DEF CloseNutGun(nutweldINFO :IN )
   ;FOLD Details
      ;FOLD Declaration
         DECL NutWeldDAT nutweldINFO
         BOOL bSkipGunChk, bSkipNutChk, bNutPresent, bMsgRelease
      ;ENDFOLD (Declaration)
      ;FOLD Implementation
         bSkipGunChk=FALSE
         bSkipNutChk=FALSE
         bNutPresent=FALSE
         bMsgRelease=FALSE
         dopw_NutIntensify(nutweldINFO.GunNr,FALSE)
         IF (bNutWeldWOJoining==FALSE) THEN
            dopw_GunWork(nutweldINFO.GunNr,TRUE)
            CONTINUE
            IF NOT (bSavedCurrentValue1 AND bSavedCurrentValue2 AND bSavedCurrentValue3) THEN
               SWITCH nutweldINFO.GunNr
                  CASE 1
                     IF NOT bSavedCurrentValue1 THEN
                        WAIT FOR bSavedCurrentValue1
                        rSetUpperLVDT_CLS_W_NUT[1] = aipw1_LVDT
                        rSetLowerLVDT_CLS_W_NUT[1] = aiNutSensorPW1
                        bSavedCurrentValue1        = TRUE
                     ENDIF
                  CASE 2
                     IF NOT bSavedCurrentValue2 THEN
                        WAIT FOR bSavedCurrentValue2
                        rSetUpperLVDT_CLS_W_NUT[2] = aipw2_LVDT
                        rSetLowerLVDT_CLS_W_NUT[2] = aiNutSensorPW2
                        bSavedCurrentValue2        = TRUE
                     ENDIF
                  CASE 3
                     IF NOT bSavedCurrentValue3 THEN
                        WAIT FOR bSavedCurrentValue3
                        rSetUpperLVDT_CLS_W_NUT[3] = aipw3_LVDT
                        rSetLowerLVDT_CLS_W_NUT[3] = aiNutSensorPW3
                        bSavedCurrentValue3        = TRUE
                     ENDIF
               ENDSWITCH
            ENDIF
            ;FOLD Gun Check
               $TIMER_STOP[nNutWeldSignalTmr]=TRUE
               $TIMER[nNutWeldSignalTmr]=nNutWeld_Signal_Timeout*(-1)
               $TIMER_STOP[nNutWeldSignalTmr]=FALSE
               WAIT FOR (((bpw_GunAtHome(nutweldINFO.GunNr)==FALSE) AND (bpw_GunAtWork(nutweldINFO.GunNr)==TRUE)) OR ($TIMER_FLAG[nNutWeldSignalTmr]==TRUE))
               $TIMER_STOP[nNutWeldSignalTmr]=TRUE
               IF (((bpw_GunAtHome(nutweldINFO.GunNr) == TRUE) OR (bpw_GunAtWork(nutweldINFO.GunNr) == FALSE)) AND (nDumpNutRetries <= nMaxDumpNutRetries)) THEN
                  bDump_Nut = TRUE
                  eCurrentState=#ERRORCloseGun
               ENDIF
               WHILE ((bNutWeldWOJoining==FALSE) AND ((bpw_GunAtHome(nutweldINFO.GunNr)==TRUE) OR (bpw_GunAtWork(nutweldINFO.GunNr)==FALSE)) AND (bSkipGunChk==FALSE) AND (nDumpNutRetries > nMaxDumpNutRetries))
                  ;FOLD Dialog "Nut Welder Open Switch Fault?"
                     REPEAT
                        nNutWeld_Handle = Set_KrlDlg (NutWeld_Msg[10], NutWeld_MsgPar[], NutWeld_SK_RetrySkip[], NutWeld_MsgOpt_Stop)
                        IF (nNutWeld_Handle > 0) THEN
                           WHILE (Exists_KrlDlg(nNutWeld_Handle, nNutWeld_Key))
                              WAIT SEC 0.024
                           ENDWHILE
                           SWITCH nNutWeld_Key
                              CASE 1 ; Diagnostic
                                 nNutWeld_Handle = Set_Krlmsg (#QUIT, NutWeld_Msg[2], NutWeld_MsgPar[], NutWeld_MsgOpt_Stop)
                                 WHILE (Exists_KrlMsg(nNutWeld_Handle))
                                    WAIT SEC 0.024
                                 ENDWHILE
                              CASE 2 ; Retry
                                 dopw_GunWork(nutweldINFO.GunNr,FALSE)
                                 WAIT SEC 1.0
                                 dopw_GunWork(nutweldINFO.GunNr,TRUE)
                                 $TIMER_STOP[nNutWeldSignalTmr]=TRUE
                                 $TIMER[nNutWeldSignalTmr]=nNutWeld_Signal_Timeout*(-1)
                                 $TIMER_STOP[nNutWeldSignalTmr]=FALSE
                                 WAIT FOR (((bpw_GunAtHome(nutweldINFO.GunNr)==FALSE) AND (bpw_GunAtWork(nutweldINFO.GunNr)==TRUE)) OR ($TIMER_FLAG[nNutWeldSignalTmr]==TRUE))
                                 $TIMER_STOP[nNutWeldSignalTmr]=TRUE
                                 bMsgRelease=TRUE
                              CASE 3 ; Skip
                                 WAIT SEC 0.100
                                 bMsgRelease=TRUE
                                 bSkipGunChk=TRUE
                           ENDSWITCH
                        ENDIF
                     UNTIL (bMsgRelease==TRUE)
                     bMsgRelease=FALSE
                  ;ENDFOLD (Dialog)
               ENDWHILE
            ;ENDFOLD (Gun Check)
            IF (PNWStyle==#STUDWELD) THEN
               dopw_StudStripped(nutweldINFO.GunNr,TRUE)
               dopw_StartFeed(nutweldINFO.GunNr,FALSE)
               ;FOLD Wait DI dipw_SpearHome==TRUE
                  $TIMER_STOP[nNutWeldSignalTmr]=TRUE
                  $TIMER[nNutWeldSignalTmr]=nNutWeld_Signal_Timeout*(-1)
                  $TIMER_STOP[nNutWeldSignalTmr]=FALSE
                  WAIT FOR ((dipw_SpearHome(nutweldINFO.GunNr)==TRUE) OR ($TIMER_FLAG[nNutWeldSignalTmr]==TRUE))
                  $TIMER_STOP[nNutWeldSignalTmr]=TRUE
               ;ENDFOLD (WaitDI dipw_SpearHome==TRUE)
            ENDIF
         ENDIF
      ;ENDFOLD (Implementation)
   ;ENDFOLD (Details)
END ; (CloseNutGun)

DEF CheckNutPresent(nutweldINFO :IN)
   ;FOLD Details
      ;FOLD Declaration
         DECL NutWeldDAT nutweldINFO
         DECL BOOL bNutChkComplete
         DECL BOOL bSkipNutChk
         DECL BOOL bInRetry
         DECL BOOL bMsgRelease
         DECL BOOL bToleranceWindowOK
         DECL REAL rSensorSample
         DECL REAL rLVDTSample
      ;ENDFOLD (Declaration)
      ;FOLD Implementation
         bMsgRelease=FALSE
         bNutChkComplete=FALSE
         bSkipNutChk=FALSE
         bInRetry=FALSE
         bToleranceWindowOK=FALSE
         WAIT FOR NOT bByPassSmartelec
         IF (bByPassSmartelec == TRUE) THEN
            RETURN ; Exit without checking
         ENDIF
         IF ((bNutWeldWOJoining==TRUE) OR (bPNWBlockFeed==TRUE)) THEN
            WAIT SEC 0.15
            RETURN ; Exit after check delay
         ENDIF
         nFeedRetries=0
         REPEAT
            bNutChkComplete=FALSE
            bInRetry=FALSE
            WAIT FOR ((rHighTolInUse-rLowTolInUse)>0) AND ((rHighTolInUse-rLowTolInUse)<1750)
            WAIT FOR ((rHighLVDTTolInUse-rLowLVDTTolInUse)>0) AND ((rHighLVDTTolInUse-rLowLVDTTolInUse)<1750)
            WAIT FOR ((rLowTolInUse)>0)
            WAIT FOR ((rHighTolInUse)>0)
            WAIT FOR ((rLowLVDTTolInUse)>0)
            WAIT FOR ((rHighLVDTTolInUse)>0)
            CloseNutGun(nutweldINFO)
            SensorSettle(nutweldINFO)
            rSensorSample=ABS(aiNutSensor(nutweldINFO.GunNr))   ; lower LVDT
            rLVDTSample=ABS(aiLVDTSensor(nutweldINFO.GunNr))    ; upper LVDT
            IF ((rSensorSample >= rLowTolInUse) AND (rSensorSample <= rHighTolInUse) AND (rLVDTSample >= rLowLVDTTolInUse) AND (rLVDTSample <= rHighLVDTTolInUse))  THEN
               bSkipNutChk=TRUE   ; do not check missing or inverted Nut if within range!
               ;save rSensorSample
               rNutSaveCount=rNutSaveCount+1
               IF (rNutSaveCount<1)OR (rNutSaveCount>50) THEN
                  rNutSaveCount=1
               ENDIF
               rNutSaveValue[rNutSaveCount]=rSensorSample
               rLVDTSaveValue[rNutSaveCount]=rLVDTSample
            ENDIF
            ;FOLD Nut Check Sequence
               ;FOLD Check for Inverted Nut
                  IF (((rSensorSample >= rHighTolInUse) OR (rLVDTSample < rLowLVDTTolInUse) OR (rLVDTSample > rHighLVDTTolInUse)) AND (nDumpNutRetries <= nMaxDumpNutRetries)) THEN
                     bDump_Nut=TRUE
                     eCurrentState=#ERRORInvertedNut
                     bNutChkComplete=FALSE
                  ENDIF
                  IF ((bSkipNutChk==FALSE) AND (bInRetry==FALSE) AND (nDumpNutRetries > nMaxDumpNutRetries)) THEN
                     IF ((rSensorSample >= rHighTolInUse) OR (rLVDTSample < rLowLVDTTolInUse) OR (rLVDTSample > rHighLVDTTolInUse)) THEN
                        ;FOLD Dialog "Nut Inverted Fault!  Press SKIP to Ignore Or Retry to Open and Close the Gun."
                           REPEAT
                              nNutWeld_Handle = Set_KrlDlg (NutWeld_Msg[48], NutWeld_MsgPar[], NutWeld_SK_RetrySkip[], NutWeld_MsgOpt_Stop)
                              IF (nNutWeld_Handle > 0) THEN
                                 WHILE (Exists_KrlDlg(nNutWeld_Handle, nNutWeld_Key))
                                    IF ($ERR.Int_Prio>0) THEN
                                       BRAKE
                                    ENDIF
                                    WAIT SEC 0.024
                                 ENDWHILE
                                 SWITCH nNutWeld_Key
                                    CASE 1 ; Diagnostic
                                       nNutWeld_Handle = Set_Krlmsg (#QUIT, NutWeld_Msg[2], NutWeld_MsgPar[], NutWeld_MsgOpt_Stop)
                                       WHILE (Exists_KrlMsg(nNutWeld_Handle))
                                          WAIT SEC 0.024
                                       ENDWHILE
                                    CASE 2 ; Retry
                                       bMsgRelease=TRUE
                                       bNutChkComplete=FALSE
                                       bInRetry=TRUE
                                       dopw_GunWork(nutweldINFO.GunNr,FALSE)
                                       WAIT SEC 1.5
                                       IF (($MODE_OP==#T1) OR ($MODE_OP==#T2)) THEN
                                          HALT
                                       ENDIF
                                    CASE 3 ; Skip
                                       WAIT SEC 0.100
                                       bMsgRelease=TRUE
                                       bSkipNutChk=TRUE
                                 ENDSWITCH
                              ENDIF
                           UNTIL (bMsgRelease==TRUE)
                           bMsgRelease=FALSE
                        ;ENDFOLD (Dialog)
                     ENDIF
                  ENDIF
               ;ENDFOLD (Check for Inverted Nut)
               ;FOLD Check for Nut Missing, If No Nut - Open Gun and feed new nut
                  IF ((bSkipNutChk==FALSE) AND (bInRetry==FALSE)) THEN
                     rSensorSample=ABS(aiNutSensor(nutweldINFO.GunNr))
                     IF ((rSensorSample <= rLowTolInUse) AND (nDumpNutRetries <= nMaxDumpNutRetries)) THEN
                        bDump_Nut=TRUE
                        eCurrentState=#ERRORNoNut
                        bNutChkComplete=FALSE
                     ENDIF
                     IF ((rSensorSample <= rLowTolInUse) AND (nDumpNutRetries > nMaxDumpNutRetries)) THEN
                        ;FOLD Dialog "Nut Not Detected Fault!  Press SKIP to Ignore Or Retry to Refeed a Nut."
                           REPEAT
                              nNutWeld_Handle = Set_KrlDlg (NutWeld_Msg[13], NutWeld_MsgPar[], NutWeld_SK_RetrySkip[], NutWeld_MsgOpt_Stop)
                              IF (nNutWeld_Handle > 0) THEN
                                 WHILE (Exists_KrlDlg(nNutWeld_Handle, nNutWeld_Key))
                                    IF ($ERR.Int_Prio>0) THEN
                                       BRAKE
                                    ENDIF
                                    WAIT SEC 0.024
                                 ENDWHILE
                                 SWITCH nNutWeld_Key
                                    CASE 1 ; Diagnostic
                                       nNutWeld_Handle = Set_Krlmsg (#QUIT, NutWeld_Msg[2], NutWeld_MsgPar[], NutWeld_MsgOpt_Stop)
                                       WHILE (Exists_KrlMsg(nNutWeld_Handle))
                                          WAIT SEC 0.024
                                       ENDWHILE
                                    CASE 2 ; Retry
                                       bMsgRelease=TRUE
                                       bNutChkComplete=FALSE
                                       bInRetry=TRUE
                                       nFeedRetries=0
                                       OpenNutGun(nutweldINFO)
                                       FeedNutReq(nutweldINFO)
                                    CASE 3 ; Skip
                                       WAIT SEC 0.100
                                       bSkipNutChk=TRUE
                                       bMsgRelease=TRUE
                                 ENDSWITCH
                              ENDIF
                           UNTIL (bMsgRelease==TRUE)
                           bMsgRelease=FALSE
                        ;ENDFOLD (Dialog)
                     ENDIF
                  ENDIF
               ;ENDFOLD (Check for Nut Missing, If No Nut - Open Gun and feed new nut)
            ;ENDFOLD (Nut Check Sequence)
         UNTIL ((bNutChkComplete==TRUE)  OR  (bSkipNutChk==TRUE) OR (bDump_Nut==TRUE))
      ;ENDFOLD (Implementation)
   ;ENDFOLD (Details)
END ; (CheckNutPresent)

;move to Reload position
GLOBAL DEF Nut_ToReloadPos(WeldPos:IN, WeldBase:IN, EnableReload:IN, Move1:IN, Move2:IN, Move3:IN, ReloadPos1:IN, ReloadPos2:IN, ReloadPos3:IN, ReloadBase1:IN, ReloadBase2:IN, ReloadBase3:IN)
   INT EnableReload
   E6POS WeldPos,ReloadPos1,ReloadPos2,ReloadPos3
   DECL FDAT WeldBase,ReloadBase1,ReloadBase2,ReloadBase3
   DECL Nut_Dump_Move Move1,Move2,Move3

   SWITCH (EnableReload)
      CASE 1
         Nut_ReLoad(Move1,ReloadPos1,ReloadBase1,FALSE)
      CASE 2
         Nut_ReLoad(Move1,ReloadPos1,ReloadBase1,FALSE)
         Nut_ReLoad(Move2,ReloadPos2,ReloadBase2,FALSE)
      CASE 3
         Nut_ReLoad(Move1,ReloadPos1,ReloadBase1,FALSE)
         Nut_ReLoad(Move2,ReloadPos2,ReloadBase2,TRUE)
         Nut_ReLoad(Move3,ReloadPos3,ReloadBase3,FALSE)
   ENDSWITCH
   WAIT FOR $IN[1025]

END

;move to Weld position
GLOBAL DEF Nut_ToWeldPos(WeldPos:IN, WeldBase:IN, EnableReload:IN, Move1:IN, Move2:IN, Move3:IN, ReloadPos1:IN, ReloadPos2:IN, ReloadPos3:IN, ReloadBase1:IN, ReloadBase2:IN, ReloadBase3:IN)
   INT EnableReload
   E6POS WeldPos,ReloadPos1,ReloadPos2,ReloadPos3
   DECL FDAT WeldBase,ReloadBase1,ReloadBase2,ReloadBase3
   DECL Nut_Dump_Move Move1,Move2,Move3

   SWITCH (EnableReload)
      CASE 1
         Nut_ReLoad(Move1,WeldPos,WeldBase,FALSE)
      CASE 2
         Nut_ReLoad(Move2,ReloadPos1,ReloadBase1,TRUE)
         Nut_ReLoad(Move1,WeldPos,WeldBase,FALSE)
      CASE 3
         Nut_ReLoad(Move3,ReloadPos2,ReloadBase2,TRUE)
         Nut_ReLoad(Move2,ReloadPos1,ReloadBase1,TRUE)
         Nut_ReLoad(Move1,WeldPos,WeldBase,FALSE)
   ENDSWITCH
   WAIT FOR $IN[1025]

END

;only for move to Reload Pos at block selection
GLOBAL DEF Nut_ReloadPos(Move1:IN, ReloadPos:IN)
   E6POS ReloadPos
   DECL Nut_Dump_Move Move1

   IF ($Mode_OP==#T1)THEN
      IF ($MOVE_BCO) THEN
         nNutWeld_Handle_SPS=Set_Krlmsg (#NOTIFY, NutWeld_Msg[61], NutWeld_MsgPar[], NutWeld_MsgOpt_NoStop)
         IF Move1==#Reload_PTP THEN
            PTP ReloadPos
         ELSE
            LIN ReloadPos
         ENDIF
         nNutWeld_Handle_SPS=Set_Krlmsg (#NOTIFY, NutWeld_Msg[62], NutWeld_MsgPar[], NutWeld_MsgOpt_NoStop)
      ENDIF
   ENDIF

END

GLOBAL DEF Nut_ReLoad(Drive:IN, ReloadPos:IN, ReloadBase:IN, Cont:IN)
   E6POS ReloadPos
   DECL FDAT ReloadBase
   DECL Nut_Dump_Move Drive
   BOOL Cont

   IF Drive==#Reload_PTP THEN
      PDAT_ACT=nut_PRELOAD
      FDAT_ACT=ReloadBase
      BAS(#PTP_PARAMS,nut_PRELOAD.VEL)
      IF Cont THEN
         PTP ReloadPos C_DIS
      ELSE
         PTP ReloadPos
      ENDIF
   ELSE ;#Reload_LIN
      LDAT_ACT=nut_LCRELOAD
      FDAT_ACT=ReloadBase
      BAS(#CP_PARAMS,nut_LCRELOAD.VEL)
      IF Cont THEN
         LIN ReloadPos C_DIS C_DIS
      ELSE
         LIN ReloadPos
      ENDIF
   ENDIF

END

DEF IntensfNutGun(nutweldINFO :IN )
   ;FOLD Details
      ;FOLD Declaration
         DECL NutWeldDAT nutweldINFO
         DECL BOOL bMsgRelease
         DECL BOOL bPreChkSkp
         DECL BOOL bIntensfChkSkp
      ;ENDFOLD (Declaration)
      ;FOLD Implementation
         bMsgRelease=FALSE
         bPreChkSkp=FALSE
         bIntensfChkSkp=FALSE
         IF (bNutWeldWOJoining==FALSE) THEN
            ;FOLD TimeOut Setup
               $TIMER_STOP[nNutWeldSignalTmr]=TRUE
               $TIMER[nNutWeldSignalTmr]=nNutWeld_Signal_Timeout*(-1)
               $TIMER_STOP[nNutWeldSignalTmr]=FALSE
            ;ENDFOLD (TimeOut Setup)
            WAIT FOR ((dipw_IntensfPresOk(nutweldINFO.GunNr)==FALSE) OR ($TIMER_FLAG[nNutWeldSignalTmr]==TRUE))
            $TIMER_STOP[nNutWeldSignalTmr]=TRUE
            WHILE ((dipw_IntensfPresOk(nutweldINFO.GunNr)==TRUE) AND (bPreChkSkp==FALSE))
               ;FOLD Dialog "Nut Welder Intensify Pressure Fault!  Pressure Switch Remained On From Last Cycle!"
                  REPEAT
                     nNutWeld_Handle = Set_KrlDlg (NutWeld_Msg[17], NutWeld_MsgPar[], NutWeld_SK_RetrySkip[], NutWeld_MsgOpt_Stop)
                     IF (nNutWeld_Handle > 0) THEN
                        WHILE (Exists_KrlDlg(nNutWeld_Handle, nNutWeld_Key))
                           IF ($ERR.Int_Prio>0) THEN
                              BRAKE
                           ENDIF
                           WAIT SEC 0.024
                        ENDWHILE
                        SWITCH nNutWeld_Key
                           CASE 1 ; Diagnostic
                              nNutWeld_Handle = Set_Krlmsg (#QUIT, NutWeld_Msg[2], NutWeld_MsgPar[], NutWeld_MsgOpt_Stop)
                              WHILE (Exists_KrlMsg(nNutWeld_Handle))
                                 WAIT SEC 0.024
                              ENDWHILE
                           CASE 2 ; Retry
                              bMsgRelease=TRUE
                           CASE 3 ; Skip
                              WAIT SEC 0.100
                              bMsgRelease=TRUE
                              bPreChkSkp=TRUE
                        ENDSWITCH
                     ENDIF
                  UNTIL (bMsgRelease==TRUE)
                  bMsgRelease=FALSE
               ;ENDFOLD (Dialog)
            ENDWHILE
            dopw_BlowOff(nutweldINFO.GunNr,TRUE)
            dopw_StudStripped(nutweldINFO.GunNr,FALSE)
            dopw_NutIntensify(nutweldINFO.GunNr, TRUE)
            ;FOLD TimeOut Setup
               $TIMER_STOP[nNutWeldSignalTmr]=TRUE
               $TIMER[nNutWeldSignalTmr]=nNutWeld_Signal_Timeout*(-1)
               $TIMER_STOP[nNutWeldSignalTmr]=FALSE
               WAIT FOR ((dipw_IntensfPresOk(nutweldINFO.GunNr)==TRUE) OR ($TIMER_FLAG[nNutWeldSignalTmr]==TRUE))
               $TIMER_STOP[nNutWeldSignalTmr]=TRUE
               WHILE ((dipw_IntensfPresOk(nutweldINFO.GunNr)==FALSE) AND (bIntensfChkSkp==FALSE))
                  ;FOLD Dialog "Nut Welder Intensify Pressure Fault!  Pressure Switch Is Not On!"
                     eCurrentState=#ERRORIntensifyWelder
                     REPEAT
                        nNutWeld_Handle = Set_KrlDlg (NutWeld_Msg[18], NutWeld_MsgPar[], NutWeld_SK_RetrySkip[], NutWeld_MsgOpt_Stop)
                        IF (nNutWeld_Handle > 0) THEN
                           WHILE (Exists_KrlDlg(nNutWeld_Handle, nNutWeld_Key))
                              IF ($ERR.Int_Prio>0) THEN
                                 BRAKE
                              ENDIF
                              WAIT SEC 0.024
                           ENDWHILE
                           SWITCH nNutWeld_Key
                              CASE 1 ; Diagnostic
                                 nNutWeld_Handle = Set_Krlmsg (#QUIT, NutWeld_Msg[2], NutWeld_MsgPar[], NutWeld_MsgOpt_Stop)
                                 WHILE (Exists_KrlMsg(nNutWeld_Handle))
                                    WAIT SEC 0.024
                                 ENDWHILE
                              CASE 2 ; Retry
                                 bMsgRelease=TRUE
                              CASE 3 ; Skip
                                 WAIT SEC 0.100
                                 bMsgRelease=TRUE
                                 bIntensfChkSkp=TRUE
                           ENDSWITCH
                        ENDIF
                     UNTIL (bMsgRelease==TRUE)
                     bMsgRelease=FALSE
                  ;ENDFOLD (Dialog)
               ENDWHILE

            ;ENDFOLD (TimeOut Setup)
         ENDIF
      ;ENDFOLD (Implementation)
   ;ENDFOLD (Details)
END ; (IntensfNutGun)

DEF WeldInitiate(nutweldINFO :IN )
   ;FOLD Details
      ;FOLD Declaration
         DECL NutWeldDAT nutweldINFO
         DECL BOOL bSkipWeld
         DECL BOOL bWeldComplete
         DECL BOOL bMsgRelease
      ;ENDFOLD (Declaration)
      ;FOLD Implementation
         bMsgRelease=FALSE
         bSkipWeld=FALSE
         ;FOLD Check the Water Flow
            WHILE NOT (di474WaterOk OR di522WaterOk OR di570WaterOk)
               IF NOT di474WaterOk THEN
                  $LOOP_MSG[] = " No WaterFlow in Gun1                                                                                                  "
               ENDIF
               IF NOT di522WaterOk THEN
                  $LOOP_MSG[] = " No WaterFlow in Gun2                                                                                                  "
               ENDIF
               IF NOT di570WaterOk THEN
                  $LOOP_MSG[] = " No WaterFlow in Gun3                                                                                                  "
               ENDIF
            ENDWHILE
            $LOOP_MSG[] = "                                                                                                                    "
         ;ENDFOLD (Check the Water Flow )
         ;FOLD Check the Temperature Water
            WHILE NOT (di472WaterTempOK OR di520WaterTempOK OR di568WaterTempOK)
               IF NOT di472WaterTempOK THEN
                  $LOOP_MSG[] = " No WaterTemp in Gun1                                                                                                  "
               ENDIF
               IF NOT di520WaterTempOK THEN
                  $LOOP_MSG[] = " No WaterTemp in Gun2                                                                                                  "
               ENDIF
               IF NOT di568WaterTempOK THEN
                  $LOOP_MSG[] = " No WaterTemp in Gun3                                                                                                  "
               ENDIF
            ENDWHILE
            $LOOP_MSG[] = "                                                                                                                    "
         ;ENDFOLD (Check the Temperature Water)
         IF (bNutWeld_InhibitWeld==TRUE) THEN
            RETURN
         ENDIF
         IF (bNutWeldWOJoining==FALSE) THEN
            REPEAT
               bWeldComplete=TRUE
               $TIMER_STOP[nNutWeldSignalTmr]=TRUE
               $TIMER[nNutWeldSignalTmr]=nNutWeld_Weld_Timeout*(-1000)
               $TIMER_STOP[nNutWeldSignalTmr]=FALSE
               dopw_WeldInit(nutweldINFO.GunNr,TRUE)
               WAIT FOR ((dipw_WeldComplete(nutweldINFO.GunNr)==TRUE) OR ($TIMER_FLAG[nNutWeldSignalTmr]==TRUE))
               $TIMER_STOP[nNutWeldSignalTmr]=TRUE

               IF (dipw_WeldComplete(nutweldINFO.GunNr)) THEN   ;count 1 weld up
                  AC_Process_Count(#Count1up)
               ENDIF

               IF ((dipw_WeldComplete(nutweldINFO.GunNr)==FALSE)) THEN
                  dopw_WeldInit(nutweldINFO.GunNr,FALSE)
                  bWeldComplete=FALSE
                  nWeldRetries = nWeldRetries + 1
                  IF (nWeldRetries > nMaxWeldRetries) then
                     do004ProcessFault=TRUE
                     ;FOLD Dialog "WELD NOT COMPLETE! Mark part as scrap, scrap part at end of cycle"
                        REPEAT
                           nNutWeld_Handle = Set_KrlDlg (NutWeld_Msg[19], NutWeld_MsgPar[], NutWeld_SK_OK[], NutWeld_MsgOpt_Stop)
                           IF (nNutWeld_Handle > 0) THEN
                              WHILE (Exists_KrlDlg(nNutWeld_Handle, nNutWeld_Key))
                                 WAIT SEC 0.024
                              ENDWHILE
                              SWITCH nNutWeld_Key
                                 CASE 1 ; Skip
                                    bWeldComplete=FALSE
                                    bMsgRelease=TRUE
                                    bSkipWeld=TRUE
                              ENDSWITCH
                              do004ProcessFault=FALSE
                           ENDIF
                        UNTIL (bMsgRelease==TRUE)
                        bMsgRelease=FALSE
                     ;ENDFOLD (Dialog)
                  ENDIF
               ENDIF
            UNTIL ((bWeldComplete==TRUE) OR (bSkipWeld==TRUE))
            bSkipWeld=FALSE
         ENDIF
         dopw_WeldInit(nutweldINFO.GunNr,FALSE)
      ;ENDFOLD (Implementation)
   ;ENDFOLD (Details)
END ; (WeldInitiate)

DEF FeedNutReq(nutweldINFO :IN)
   ;FOLD Details
      ;FOLD Declaration
         DECL NutWeldDAT nutweldINFO
         DECL BOOL bSkipPinRet
         DECL BOOL bMsgRelease
         DECL BOOL bSkipFeed
      ;ENDFOLD (Declaration)
      ;FOLD Implementation
         bSkipPinRet=FALSE
         bMsgRelease=FALSE
         bSkipFeed=FALSE
         IF ((bNutWeldWOJoining==TRUE) OR (bPNWBlockFeed==TRUE)) THEN
            WAIT SEC 0.15
            RETURN ; Exit after check delay
         ENDIF
         ;FOLD Check that the Locate Pin is Advanced
            dopw_PinAdv(nutweldINFO.GunNr, TRUE)
            $TIMER_STOP[nNutWeldSignalTmr]=TRUE
            $TIMER[nNutWeldSignalTmr]=nNutWeld_Signal_Timeout*(-1)
            $TIMER_STOP[nNutWeldSignalTmr]=FALSE
            WAIT FOR ((dipw_PinReturn(nutweldINFO.GunNr)==FALSE) OR ($TIMER_FLAG[nNutWeldSignalTmr]==TRUE)) ; Convert to no nut analog
            $TIMER_STOP[nNutWeldSignalTmr]=TRUE
            ; Modified for nutweld specific, original refernce was studweld
            WHILE ((dipw_PinReturn(nutweldINFO.GunNr)==TRUE) AND (bSkipPinRet==FALSE))
               ;FOLD Dialog "Welder Pin is Not Advanced!  Check the Pin or Smart Electrode!"
                  REPEAT
                     nNutWeld_Handle = Set_KrlDlg (NutWeld_Msg[15], NutWeld_MsgPar[], NutWeld_SK_RetrySkip[], NutWeld_MsgOpt_Stop)
                     IF (nNutWeld_Handle > 0) THEN
                        WHILE (Exists_KrlDlg(nNutWeld_Handle, nNutWeld_Key))
                           WAIT SEC 0.024
                        ENDWHILE
                        SWITCH nNutWeld_Key
                           CASE 1 ; Diagnostic
                              nNutWeld_Handle = Set_Krlmsg (#QUIT, NutWeld_Msg[2], NutWeld_MsgPar[], NutWeld_MsgOpt_Stop)
                              WHILE (Exists_KrlMsg(nNutWeld_Handle))
                                 WAIT SEC 0.024
                              ENDWHILE
                           CASE 2 ; Retry
                              bMsgRelease=TRUE
                           CASE 3 ; Skip
                              bMsgRelease=TRUE
                              bSkipPinRet=TRUE
                        ENDSWITCH
                     ENDIF
                  UNTIL (bMsgRelease==TRUE)
                  bMsgRelease=FALSE
               ;ENDFOLD (Dialog)
            ENDWHILE
         ;ENDFOLD (Check that the Locate Pin is Advanced)
         dopw_StartFeed(nutweldINFO.GunNr,TRUE)
         ;FOLD WaitDI dipw_SpearHome==FALSE
            $TIMER_STOP[nNutWeldSignalTmr]=TRUE
            $TIMER[nNutWeldSignalTmr]=nNutWeld_Signal_Timeout*(-1)
            $TIMER_STOP[nNutWeldSignalTmr]=FALSE
            WAIT FOR ((dipw_SpearHome(nutweldINFO.GunNr)==FALSE) OR ($TIMER_FLAG[nNutWeldSignalTmr]==TRUE))
            $TIMER_STOP[nNutWeldSignalTmr]=TRUE
         ;ENDFOLD (WaitDI dipw_SpearHome==FALSE)
         IF (PNWStyle==#NUTWELD) THEN
            ;FOLD WaitDI dipw_SpearHome==TRUE
               $TIMER_STOP[nNutWeldSignalTmr]=TRUE
               $TIMER[nNutWeldSignalTmr]=nNutWeld_Signal_Timeout*(-1)
               $TIMER_STOP[nNutWeldSignalTmr]=FALSE
               WAIT FOR ((dipw_SpearHome(nutweldINFO.GunNr)==TRUE) OR ($TIMER_FLAG[nNutWeldSignalTmr]==TRUE))
               $TIMER_STOP[nNutWeldSignalTmr]=TRUE
            ;ENDFOLD (WaitDI dipw_SpearHome==TRUE)
         ENDIF
         ;FOLD WaitDI dipw_FeedComplt==TRUE
            $TIMER_STOP[nNutWeldFeedTmr]=TRUE
            $TIMER[nNutWeldFeedTmr]=nNutWeld_Feed_Timeout*(-3000)
            $TIMER_STOP[nNutWeldFeedTmr]=FALSE
            WAIT FOR ((dipw_FeedComplt(nutweldINFO.GunNr)==TRUE) OR ($TIMER_FLAG[nNutWeldFeedTmr]==TRUE))
            $TIMER_STOP[nNutWeldFeedTmr]=TRUE
            WHILE ((dipw_FeedComplt(nutweldINFO.GunNr)==FALSE) AND (bSkipFeed==FALSE))
               ;FOLD Dialog "Feed Request Timeout Fault!  Check the Bowl Feeder!"
                  REPEAT
                     nNutWeld_Handle = Set_KrlDlg (NutWeld_Msg[49], NutWeld_MsgPar[], NutWeld_SK_RetrySkip[], NutWeld_MsgOpt_Stop)
                     IF (nNutWeld_Handle > 0) THEN
                        WHILE (Exists_KrlDlg(nNutWeld_Handle, nNutWeld_Key))
                           WAIT SEC 0.024
                        ENDWHILE
                        SWITCH nNutWeld_Key
                           CASE 1 ; Diagnostic
                              nNutWeld_Handle = Set_Krlmsg (#QUIT, NutWeld_Msg[2], NutWeld_MsgPar[], NutWeld_MsgOpt_Stop)
                              WHILE (Exists_KrlMsg(nNutWeld_Handle))
                                 WAIT SEC 0.024
                              ENDWHILE
                           CASE 2 ; Retry
                              bMsgRelease=TRUE
                              dopw_StartFeed(nutweldINFO.GunNr,FALSE)
                              WAIT SEC 1
                              dopw_StartFeed(nutweldINFO.GunNr,TRUE)
                              WAIT SEC 2
                           CASE 3 ; Skip
                              bMsgRelease=TRUE
                              bSkipFeed=TRUE
                        ENDSWITCH
                     ENDIF
                  UNTIL (bMsgRelease==TRUE)
                  bMsgRelease=FALSE
               ;ENDFOLD (Dialog)
            ENDWHILE
         ;ENDFOLD (WaitDI dipw_FeedComplt==TRUE)
         IF (PNWStyle==#NUTWELD) THEN
            dopw_StartFeed(nutweldINFO.GunNr,FALSE)
         ENDIF
      ;ENDFOLD (Implementation)
   ;ENDFOLD (Details)
END ; (FeedNutReq)

DEF SensorSettle(nutweldINFO :IN )
   ;FOLD Details
      ;FOLD Declaration
         DECL NutWeldDAT nutweldINFO
         REAL rPrimaryValue, rSecondaryValue, rSensorSample
      ;ENDFOLD (Declaration)
      ;FOLD Implementation
         REPEAT
            rPrimaryValue = ABS(aiNutSensor(nutweldINFO.GunNr))
            WAIT SEC rSensorSettleTime
            rSecondaryValue = ABS(aiNutSensor(nutweldINFO.GunNr))
            IF (ABS(rPrimaryValue - rSecondaryValue) > 40) THEN
               WAIT SEC rSensorSettleTime
            ENDIF
         UNTIL (ABS(rPrimaryValue - rSecondaryValue)<20)
      ;ENDFOLD (Implementation)
   ;ENDFOLD (Details)
END ; (SensorSettle)

DEF dopw_NutIntensify(nGunNr :IN, bState :IN )
   ;FOLD Details
      ;FOLD Declaration
         DECL INT nGunNr
         DECL BOOL bState
      ;ENDFOLD (Declaration)
      ;FOLD Implementation
         SWITCH nGunNr
            CASE 1
               dopw1_Nut1Intensify_Home=NOT(bState)
               dopw1_Nut1Intensify=bState
            CASE 2
               dopw2_Nut1Intensify_Home=NOT(bState)
               dopw2_Nut1Intensify=bState
            CASE 3
               dopw3_Nut1Intensify_Home=NOT(bState)
               dopw3_Nut1Intensify=bState
         ENDSWITCH
      ;ENDFOLD (Implementation)
   ;ENDFOLD (Details)
END ; (dopw_NutIntensify)

DEF dopw_GunWork(nGunNr :IN, bState :IN )
   ;FOLD Details
      ;FOLD Declaration
         DECL INT nGunNr
         DECL BOOL bState
      ;ENDFOLD (Declaration)
      ;FOLD Implementation
         SWITCH nGunNr
            CASE 1
               dopw1_GunWork=bState
               dopw1_GunHome=NOT (bState)
               IF (bState==FALSE) THEN
                  dopw_NutIntensify(nGunNr,FALSE)
               ENDIF
            CASE 2
               dopw2_GunWork=bState
               dopw2_GunHome=NOT (bState)
               IF (bState==FALSE) THEN
                  dopw_NutIntensify(nGunNr,FALSE)
               ENDIF
            CASE 3
               dopw3_GunWork=bState
               dopw3_GunHome=NOT (bState)
               IF (bState==FALSE) THEN
                  dopw_NutIntensify(nGunNr,FALSE)
               ENDIF
         ENDSWITCH
      ;ENDFOLD (Implementation)
   ;ENDFOLD (Details)
END ; (dopw_GunWork)

DEF dopw_PinAdv(nGunNr :IN, bState :IN )
   ;FOLD Details
      ;FOLD Declaration
         DECL INT nGunNr
         DECL BOOL bState
      ;ENDFOLD (Declaration)
      ;FOLD Implementation
         SWITCH nGunNr
            CASE 1
               dopw1_AdvancePin=bState
               dopw1_ReturnPin=NOT (bState)
            CASE 2
               dopw2_AdvancePin=bState
               dopw2_ReturnPin=NOT (bState)
            CASE 3
               dopw3_AdvancePin=bState
               dopw3_ReturnPin=NOT (bState)
         ENDSWITCH
      ;ENDFOLD (Implementation)
   ;ENDFOLD (Details)
END ; (dopw_PinAdv)

DEF dopw_StepperWarningPL(nGunNr :IN, bState :IN )
   ;FOLD Details
      ;FOLD Declaration
         DECL INT nGunNr
         DECL BOOL bState
      ;ENDFOLD (Declaration)
      ;FOLD Implementation
         SWITCH nGunNr
            CASE 1
               dopw1_StepperWarningPL=bState
            CASE 2
               dopw2_StepperWarningPL=bState
            CASE 3
               dopw3_StepperWarningPL=bState
         ENDSWITCH
      ;ENDFOLD (Implementation)
   ;ENDFOLD (Details)
END ; (dopw_StepperWarningPL)

DEF dopw_EndofStepperPL(nGunNr :IN, bState :IN )
   ;FOLD Details
      ;FOLD Declaration
         DECL INT nGunNr
         DECL BOOL bState
      ;ENDFOLD (Declaration)
      ;FOLD Implementation
         SWITCH nGunNr
            CASE 1
               dopw1_EndofStepperPL=bState
            CASE 2
               dopw2_EndofStepperPL=bState
            CASE 3
               dopw3_EndofStepperPL=bState
         ENDSWITCH
      ;ENDFOLD (Implementation)
   ;ENDFOLD (Details)
END ; (dopw_EndofStepperPL)

DEF dopw_StartFeed(nGunNr :IN, bState :IN )
   ;FOLD Details
      ;FOLD Declaration
         DECL INT nGunNr
         DECL BOOL bState
      ;ENDFOLD (Declaration)
      ;FOLD Implementation
         SWITCH nGunNr
            CASE 1
               dopw1_StartFeed=bState
            CASE 2
               dopw2_StartFeed=bState
            CASE 3
               dopw3_StartFeed=bState
         ENDSWITCH
      ;ENDFOLD (Implementation)
   ;ENDFOLD (Details)
END ; (dopw_StartFeed)

DEF dopw_StartWater(nGunNr :IN, bState :IN )
   ;FOLD Details
      ;FOLD Declaration
         DECL INT nGunNr
         DECL BOOL bState
      ;ENDFOLD (Declaration)
      ;FOLD Implementation
         SWITCH nGunNr
            CASE 1
               dopw1_StartWater=bState
            CASE 2
               dopw2_StartWater=bState
            CASE 3
               dopw3_StartWater=bState
         ENDSWITCH
      ;ENDFOLD (Implementation)
   ;ENDFOLD (Details)
END ; (dopw_StartWater)

DEF dopw_SetPrgNr(nGunNr :IN, nPrgNr :IN )
   ;FOLD Details
      ;FOLD Declaration
         DECL INT nGunNr
         DECL INT nPrgNr
      ;ENDFOLD (Declaration)
      ;FOLD Implementation
         SWITCH nGunNr
            CASE 1
               gdopw1_SpotNumber=nPrgNr
            CASE 2
               gdopw2_SpotNumber=nPrgNr
            CASE 3
               gdopw3_SpotNumber=nPrgNr
         ENDSWITCH
      ;ENDFOLD (Implementation)
   ;ENDFOLD (Details)
END ; (dopw_SetPrgNr)

DEF dopw_WeldInit(nGunNr :IN, bState :IN )
   ;FOLD Details
      ;FOLD Declaration
         DECL INT nGunNr
         DECL BOOL bState
      ;ENDFOLD (Declaration)
      ;FOLD Implementation
         SWITCH nGunNr
            CASE 1
               dopw1_WeldInit=bState
            CASE 2
               dopw2_WeldInit=bState
            CASE 3
               dopw3_WeldInit=bState
         ENDSWITCH
      ;ENDFOLD (Implementation)
   ;ENDFOLD (Details)
END ; (dopw_WeldInit)

DEF dopw_FaultReset(nGunNr :IN, bState :IN )
   ;FOLD Details
      ;FOLD Declaration
         DECL INT nGunNr
         DECL BOOL bState
      ;ENDFOLD (Declaration)
      ;FOLD Implementation
         SWITCH nGunNr
            CASE 1
               dopw1_FaultReset=bState
            CASE 2
               dopw2_FaultReset=bState
            CASE 3
               dopw3_FaultReset=bState
         ENDSWITCH
      ;ENDFOLD (Implementation)
   ;ENDFOLD (Details)
END ; (dopw_FaultReset)

DEF dopw_BlowOff(nGunNr :IN, bState :IN )
   ;FOLD Details
      ;FOLD Declaration
         DECL INT nGunNr
         DECL BOOL bState
      ;ENDFOLD (Declaration)
      ;FOLD Implementation
         SWITCH nGunNr
            CASE 1
               dopw1_BlowOff=bState
            CASE 2
               dopw2_BlowOff=bState
            CASE 3
               dopw3_BlowOff=bState
         ENDSWITCH
      ;ENDFOLD (Implementation)
   ;ENDFOLD (Details)
END ; (dopw_BlowOff)

DEF dopw_StudStripped(nGunNr :IN, bState :IN )
   ;FOLD Details
      ;FOLD Declaration
         DECL INT nGunNr
         DECL BOOL bState
      ;ENDFOLD (Declaration)
      ;FOLD Implementation
         SWITCH nGunNr
            CASE 1
               dopw1_StudStripped=bState
            CASE 2
               dopw2_StudStripped=bState
            CASE 3
               dopw3_StudStripped=bState
         ENDSWITCH
      ;ENDFOLD (Implementation)
   ;ENDFOLD (Details)
END ; (dopw_StudStripped)

DEFFCT INT Get_FaultResetNr(nGunNr :IN )
   ;FOLD Details
      ;FOLD Declaration
         DECL INT nGunNr
         DECL SIGINF SignalIOInfo
      ;ENDFOLD (Declaration)
      ;FOLD Implementation
         SWITCH nGunNr
            CASE 1
               SignalIOInfo=GET_SIG_INF("dopw1_FaultReset")
               RETURN(SignalIOInfo.IDX)
            CASE 2
               SignalIOInfo=GET_SIG_INF("dopw2_FaultReset")
               RETURN(SignalIOInfo.IDX)
            CASE 3
               SignalIOInfo=GET_SIG_INF("dopw3_FaultReset")
               RETURN(SignalIOInfo.IDX)
         ENDSWITCH
      ;ENDFOLD (Implementation)
   ;ENDFOLD (Details)
ENDFCT ; (Get_FaultResetNr)

DEFFCT BOOL bpw_GunAtHome(nGunNr :IN )
   ;FOLD Details
      ;FOLD Declaration
         DECL INT nGunNr
      ;ENDFOLD (Declaration)
      ;FOLD Implementation
         SWITCH nGunNr
            CASE 1
               RETURN(bpw1_GunAtHome)
            CASE 2
               RETURN(bpw2_GunAtHome)
            CASE 3
               RETURN(bpw3_GunAtHome)
         ENDSWITCH
      ;ENDFOLD (Implementation)
   ;ENDFOLD (Details)
ENDFCT ; (bpw_GunAtHome)

DEFFCT BOOL bpw_GunAtWork(nGunNr :IN )
   ;FOLD Details
      ;FOLD Declaration
         DECL INT nGunNr
      ;ENDFOLD (Declaration)
      ;FOLD Implementation
         $OUT[148]=FALSE
         SWITCH nGunNr
            CASE 1
               RETURN(bpw1_GunAtWork)
            CASE 2
               RETURN(bpw2_GunAtWork)
            CASE 3
               RETURN(bpw3_GunAtWork)
         ENDSWITCH
      ;ENDFOLD (Implementation)
   ;ENDFOLD (Details)
ENDFCT ; (bpw_GunAtWork)

DEFFCT BOOL dipw_IntensfPresOk(nGunNr :IN )
   ;FOLD Details
      ;FOLD Declaration
         DECL INT nGunNr
      ;ENDFOLD (Declaration)
      ;FOLD Implementation
         SWITCH nGunNr
            CASE 1
               RETURN(dipw1_IntensfPresOk)
            CASE 2
               RETURN(dipw2_IntensfPresOk)
            CASE 3
               RETURN(dipw3_IntensfPresOk)
         ENDSWITCH
      ;ENDFOLD (Implementation)
   ;ENDFOLD (Details)
ENDFCT ; (dipw_IntensfPresOk)

DEFFCT BOOL dipw_StepperWarning(nGunNr :IN )
   ;FOLD Details
      ;FOLD Declaration
         DECL INT nGunNr
      ;ENDFOLD (Declaration)
      ;FOLD Implementation
         SWITCH nGunNr
            CASE 1
               RETURN(dipw1_StepperWarning)
            CASE 2
               RETURN(dipw2_StepperWarning)
            CASE 3
               RETURN(dipw3_StepperWarning)
         ENDSWITCH
      ;ENDFOLD (Implementation)
   ;ENDFOLD (Details)
ENDFCT ; (dipw_StepperWarning)

DEFFCT BOOL dipw_EndOfStepper(nGunNr :IN )
   ;FOLD Details
      ;FOLD Declaration
         DECL INT nGunNr
      ;ENDFOLD (Declaration)
      ;FOLD Implementation
         SWITCH nGunNr
            CASE 1
               RETURN(dipw1_EndOfStepper)
            CASE 2
               RETURN(dipw2_EndOfStepper)
            CASE 3
               RETURN(dipw3_EndOfStepper)
         ENDSWITCH
      ;ENDFOLD (Implementation)
   ;ENDFOLD (Details)
ENDFCT ; (dipw_EndOfStepper)

DEFFCT BOOL dipw_XtfmrTempOk(nGunNr :IN )
   ;FOLD Details
      ;FOLD Declaration
         DECL INT nGunNr
      ;ENDFOLD (Declaration)
      ;FOLD Implementation
         SWITCH nGunNr
            CASE 1
               RETURN(dipw1_XtfmrTempOk)
            CASE 2
               RETURN(dipw2_XtfmrTempOk)
            CASE 3
               RETURN(dipw3_XtfmrTempOk)
         ENDSWITCH
      ;ENDFOLD (Implementation)
   ;ENDFOLD (Details)
ENDFCT ; (dipw_XtfmrTempOk)

DEFFCT BOOL dipw_WaterOk(nGunNr :IN )
   ;FOLD Details
      ;FOLD Declaration
         DECL INT nGunNr
      ;ENDFOLD (Declaration)
      ;FOLD Implementation
         SWITCH nGunNr
            CASE 1
               RETURN(dipw1_WaterOk)
            CASE 2
               RETURN(dipw2_WaterOk)
            CASE 3
               RETURN(dipw3_WaterOk)
         ENDSWITCH
      ;ENDFOLD (Implementation)
   ;ENDFOLD (Details)
ENDFCT ; (dipw_WaterOk)

DEFFCT BOOL dipw_WaterTempOk(nGunNr :IN )
   ;FOLD Details
      ;FOLD Declaration
         DECL INT nGunNr
      ;ENDFOLD (Declaration)
      ;FOLD Implementation
         SWITCH nGunNr
            CASE 1
               RETURN(di472WaterTempOk)
            CASE 2
               RETURN(di520WaterTempOk)
            CASE 3
               RETURN(di568WaterTempOk)
         ENDSWITCH
      ;ENDFOLD (Implementation)
   ;ENDFOLD (Details)
ENDFCT ; (dipw_WaterTempOk)

DEFFCT BOOL dipw_WeldComplete(nGunNr :IN )
   ;FOLD Details
      ;FOLD Declaration
         DECL INT nGunNr
      ;ENDFOLD (Declaration)
      ;FOLD Implementation
         SWITCH nGunNr
            CASE 1
               RETURN(dipw1_WeldComplete)
            CASE 2
               RETURN(dipw2_WeldComplete)
            CASE 3
               RETURN(dipw3_WeldComplete)
         ENDSWITCH
      ;ENDFOLD (Implementation)
   ;ENDFOLD (Details)
ENDFCT ; (dipw_WeldComplete)

DEFFCT BOOL dipw_Ready(nGunNr :IN )
   ;FOLD Details
      ;FOLD Declaration
         DECL INT nGunNr
      ;ENDFOLD (Declaration)
      ;FOLD Implementation
         SWITCH nGunNr
            CASE 1
               RETURN(dipw1_Ready)
            CASE 2
               RETURN(dipw2_Ready)
            CASE 3
               RETURN(dipw3_Ready)
         ENDSWITCH
      ;ENDFOLD (Implementation)
   ;ENDFOLD (Details)
ENDFCT ; (dipw_Ready)

DEFFCT BOOL dipw_Fault(nGunNr :IN )
   ;FOLD Details
      ;FOLD Declaration
         DECL INT nGunNr
      ;ENDFOLD (Declaration)
      ;FOLD Implementation
         SWITCH nGunNr
            CASE 1
               RETURN(dipw1_Fault)
            CASE 2
               RETURN(dipw2_Fault)
            CASE 3
               RETURN(dipw3_Fault)
         ENDSWITCH
      ;ENDFOLD (Implementation)
   ;ENDFOLD (Details)
ENDFCT ; (dipw_Fault)

DEFFCT BOOL dipw_SpearHome(nGunNr :IN )
   ;FOLD Details
      ;FOLD Declaration
         DECL INT nGunNr
      ;ENDFOLD (Declaration)
      ;FOLD Implementation
         SWITCH nGunNr
            CASE 1
               RETURN(dipw1_SpearHome)
            CASE 2
               RETURN(dipw2_SpearHome)
            CASE 3
               RETURN(dipw3_SpearHome)
         ENDSWITCH
      ;ENDFOLD (Implementation)
   ;ENDFOLD (Details)
ENDFCT ; (dipw_SpearHome)

DEFFCT BOOL dipw_PinReturn(nGunNr :IN )
   ;FOLD Details
      ;FOLD Declaration
         DECL INT nGunNr
      ;ENDFOLD (Declaration)
      ;FOLD Implementation
         SWITCH nGunNr
            CASE 1
               RETURN(dipw1_PinReturn)
            CASE 2
               RETURN(dipw2_PinReturn)
            CASE 3
               RETURN(dipw3_PinReturn)
         ENDSWITCH
      ;ENDFOLD (Implementation)
   ;ENDFOLD (Details)
ENDFCT ; (dipw_PinReturn)

DEFFCT BOOL dipw_FeedComplt(nGunNr :IN )
   ;FOLD Details
      ;FOLD Declaration
         DECL INT nGunNr
      ;ENDFOLD (Declaration)
      ;FOLD Implementation
         SWITCH nGunNr
            CASE 1
               RETURN(dipw1_FeedComplt)
            CASE 2
               RETURN(dipw2_FeedComplt)
            CASE 3
               RETURN(dipw3_FeedComplt)
         ENDSWITCH
      ;ENDFOLD (Implementation)
   ;ENDFOLD (Details)
ENDFCT ; (dipw_FeedComplt)

DEFFCT REAL aiNutSensor(nGunNr :IN )
   ;FOLD Details
      ;FOLD Declaration
         DECL INT nGunNr
      ;ENDFOLD (Declaration)
      ;FOLD Implementation
         SWITCH nGunNr
            CASE 1
               RETURN(aiNutSensorPW1)
            CASE 2
               RETURN(aiNutSensorPW2)
            CASE 3
               RETURN(aiNutSensorPW3)
         ENDSWITCH
      ;ENDFOLD (Implementation)
   ;ENDFOLD (Details)
ENDFCT ; (aiNutSensor)

DEFFCT REAL aiLVDTSensor(nGunNr :IN )
   ;FOLD Details
      ;FOLD Declaration
         DECL INT nGunNr
      ;ENDFOLD (Declaration)
      ;FOLD Implementation
         SWITCH nGunNr
            CASE 1
               RETURN(aipw1_LVDT)
            CASE 2
               RETURN(aipw2_LVDT)
            CASE 3
               RETURN(aipw3_LVDT)
         ENDSWITCH
      ;ENDFOLD (Implemenation)
   ;ENDFOLD (Details)
ENDFCT ; (aiLVDTSensor)

--- nutweldroutines.dat ---
&ACCESS RVO3
&REL 3482
&PARAM DISKPATH = KRC:\R1\TP\NutWeld
DEFDAT  nutweldroutines PUBLIC
;*********************************
;* Package:     NutWeldRoutines  *
;* Release      V1.0.4           *
;* Date:        01.2016          *
;* GUI Version: > = V8.3         *
;*********************************

GLOBAL ENUM Nut_Dump_Move Reload_PTP,Reload_LIN
DECL GLOBAL BOOL bDump_Nut
DECL GLOBAL INT nMaxGunNr=3
DECL GLOBAL INT nMaxWeldRetries=0
DECL GLOBAL INT nMaxFeedRetries=0
DECL GLOBAL INT nMaxDumpNutRetries=10
DECL GLOBAL INT nSpotNrTstCrnt=255
DECL GLOBAL BOOL bPNWBlockFeed=FALSE
DECL GLOBAL INT nNutWeldSignalTmr=41
DECL GLOBAL INT nNutWeld_Signal_Timeout=6000 ; (ms)
DECL GLOBAL INT nNutWeldFeedTmr=41
DECL GLOBAL INT nNutWeld_Feed_Timeout=7 ; (s)
DECL GLOBAL INT nNutWeldWeldTmr=41
DECL GLOBAL INT nNutWeld_Weld_Timeout=8 ; (s)
DECL GLOBAL INT nNutWeldManWeldTmr=42
DECL GLOBAL INT nNutWeld_ManWeld_Timeout=5 ; (s)
DECL GLOBAL BOOL bNutWeldComplete=FALSE
DECL GLOBAL INT nNutWeld_WtrStrtTime=4 ; (s)
DECL GLOBAL REAL rSensorSettleTime=0.200000 ; (s)
DECL GLOBAL BOOL bByPassSmartelec=FALSE
DECL GLOBAL NutWeld_Style_Type PNWStyle=#NUTWELD
DECL GLOBAL BOOL bNutWeld_PreAdvPin=FALSE
;FOLD NutWeld UserKeyBar1
DECL GLOBAL BOOL bNutWeldWOJoinSTK=TRUE ; Button 1
DECL GLOBAL BOOL bNutWeldResetSTK=FALSE ; Button 4
;ENDFOLD (NutWeld UserKeyBar1)
;FOLD NutWeld UserKeyBar2
DECL GLOBAL INT nNutWeldGunNrSTK=3 ; Button 1
DECL GLOBAL BOOL bNutWeldOpnGunSTK=FALSE ; Button 2
DECL GLOBAL BOOL bNutWeldClsGunSTK=FALSE ; Button 3
DECL GLOBAL BOOL bNutWeldAdvRetPinSTK=FALSE ; Button 4
;ENDFOLD (NutWeld UserKeyBar2)
;FOLD NutWeld UserKeyBar3
; DECL GLOBAL INT nNutWeldGunNrSTK=1 ; Button 1 - Declared in UserKeyBar2
DECL GLOBAL INT nNutWeldSpotNrSTK=1 ; Button 2 - Value
DECL GLOBAL INT nNutWeldSpotMinSTK=1 ; Button 2 - Minimum
DECL GLOBAL INT nNutWeldSpotMaxSTK=999 ; Button 2 - Maximium
DECL GLOBAL BOOL bNutWeldManWeldSTK=FALSE ; Button 4
;ENDFOLD (NutWeld UserKeyBar3)
;FOLD NutWeld UserKeyBar4
; DECL GLOBAL INT nNutWeldGunNrSTK=1 ; Button 1 - Declared in UserKeyBar2
DECL GLOBAL BOOL bNutWeldTchAnlgSTK=FALSE ; Button 2
DECL GLOBAL BOOL bNutWeldAlgNoNutReq=FALSE ; Button 2-1
DECL GLOBAL BOOL bNutWeldAlgWNutReq=FALSE ; Button 2-2
DECL GLOBAL BOOL bNutWeldAlgInNutReq=FALSE ; Button 2-3
DECL GLOBAL BOOL bNutWeldAlgCheckReq=FALSE ; Button 2-4
DECL GLOBAL BOOL bNutWeldTstFrceSTK=FALSE ; Button 3
DECL GLOBAL BOOL bNutWeldTstCrntSTK=FALSE ; Button 4
;ENDFOLD (NutWeld UserKeyBar4)
;FOLD New message
DECL GLOBAL REAL rStartValue
DECL GLOBAL REAL rActualValue
DECL GLOBAL BOOL WeldTouchUp=FALSE
;ENDFOLD
;FOLD DNMP System 1 IO Data
;GLOBAL SIGNAL dipw1_Reserved $IN[465]
;GLOBAL SIGNAL dipw1_Reserved $IN[466]
;GLOBAL SIGNAL dipw1_Reserved $IN[467]
;GLOBAL SIGNAL dipw1_Reserved $IN[468]
;GLOBAL SIGNAL dipw1_Reserved $IN[469]
;GLOBAL SIGNAL dipw1_Reserved $IN[470]
;GLOBAL SIGNAL dipw1_Reserved $IN[471]
;GLOBAL SIGNAL dipw1_Reserved $IN[472]
GLOBAL SIGNAL dipw1_AirOK $IN[473]
;GLOBAL SIGNAL dipw1_WaterOk $IN[474]
GLOBAL BOOL dipw1_WaterOk=TRUE

GLOBAL SIGNAL dipw1_XtfmrTempOk $IN[475]
GLOBAL SIGNAL dipw1_GunAtHome $IN[476]
DECL GLOBAL BOOL bpw1_GunAtHome=FALSE
GLOBAL SIGNAL dipw1_GunAtWork $IN[477]
DECL GLOBAL BOOL bpw1_GunAtWork=FALSE
GLOBAL SIGNAL dipw1_PinReturn $IN[478]
GLOBAL SIGNAL dipw1_IntensfPresOk $IN[479]
GLOBAL SIGNAL dipw1_HopperLowLevel $IN[480]
GLOBAL SIGNAL dipw1_FeedComplt $IN[481]
GLOBAL SIGNAL dipw1_SpearHome $IN[482]
;GLOBAL SIGNAL dipw1_Reserved $OUT[465]
;GLOBAL SIGNAL dipw1_Reserved $OUT[466]
;GLOBAL SIGNAL dipw1_Reserved $OUT[467]
;GLOBAL SIGNAL dipw1_Reserved $OUT[468]
;GLOBAL SIGNAL dipw1_Reserved $OUT[469]
GLOBAL SIGNAL dopw1_Hidraulyc_Valve $OUT[470]
GLOBAL SIGNAL dopw1_GunHome $OUT[471] ;Nueva
GLOBAL SIGNAL dopw1_GunWork $OUT[472]
GLOBAL SIGNAL dopw1_Nut1Intensify_Home $OUT[473]
GLOBAL SIGNAL dopw1_Nut1Intensify $OUT[474]
GLOBAL SIGNAL dopw1_StartWater $OUT[475]
GLOBAL SIGNAL dopw1_StartFeed $OUT[476]
GLOBAL SIGNAL dopw1_LevelOk $OUT[477]
GLOBAL SIGNAL dopw1_LowLevel $OUT[478]
GLOBAL SIGNAL dopw1_StepperWarningPL $OUT[479]
GLOBAL SIGNAL dopw1_EndofStepperPL $OUT[480]
GLOBAL SIGNAL dopw1_BlowOff $OUT[494]
GLOBAL SIGNAL dopw1_AdvancePin $OUT[495]
GLOBAL SIGNAL dopw1_ReturnPin $OUT[496]
GLOBAL SIGNAL dopw1_StudStripped $OUT[497]
;ENDFOLD (DNMP System 1 IO Data)
;FOLD Welder System 1 IO Data
GLOBAL SIGNAL dipw1_WeldComplete $IN[483]
GLOBAL SIGNAL dipw1_Ready $IN[484]
GLOBAL SIGNAL dipw1_Fault $IN[485]
GLOBAL SIGNAL dipw1_StepperWarning $IN[486]
GLOBAL SIGNAL dipw1_EndOfStepper $IN[487]
GLOBAL SIGNAL dipw1_StepperAreReset $IN[488]
GLOBAL SIGNAL dopw1_WeldContactEnable $OUT[481]
GLOBAL SIGNAL dopw1_WeldOnExternal $OUT[482]
GLOBAL SIGNAL dopw1_WeldInit $OUT[483]
GLOBAL SIGNAL dopw1_FaultReset $OUT[484]
GLOBAL SIGNAL dopw1_StepperReset $OUT[485]
GLOBAL SIGNAL dopw1_486SpotNumber1 $OUT[486]
GLOBAL SIGNAL dopw1_487SpotNumber2 $OUT[487]
GLOBAL SIGNAL dopw1_488SpotNumber4 $OUT[488]
GLOBAL SIGNAL dopw1_489SpotNumber8 $OUT[489]
GLOBAL SIGNAL dopw1_490SpotNumber16 $OUT[490]
GLOBAL SIGNAL dopw1_491SpotNumber32 $OUT[491]
GLOBAL SIGNAL dopw1_492SpotNumber64 $OUT[492]
GLOBAL SIGNAL dopw1_493SpotNumber128 $OUT[493]
GLOBAL SIGNAL gdopw1_SpotNumber $OUT[486]  TO $OUT[493]
;ENDFOLD (Welder System 1 IO Data)
;FOLD DNMP System 2 IO Data
;GLOBAL SIGNAL dipw2_Reserved $IN[513]
;GLOBAL SIGNAL dipw2_Reserved $IN[514]
;GLOBAL SIGNAL dipw2_Reserved $IN[515]
;GLOBAL SIGNAL dipw2_Reserved $IN[516]
;GLOBAL SIGNAL dipw2_Reserved $IN[517]
;GLOBAL SIGNAL dipw2_Reserved $IN[518]
;GLOBAL SIGNAL dipw2_Reserved $IN[519]
;GLOBAL SIGNAL dipw2_Reserved $IN[520]
GLOBAL SIGNAL dipw2_AirOK $IN[521]
GLOBAL SIGNAL dipw2_WaterOk $IN[522]
GLOBAL SIGNAL dipw2_XtfmrTempOk $IN[523]
GLOBAL SIGNAL dipw2_GunAtHome $IN[524]
GLOBAL SIGNAL dipw2_GunAtWork $IN[525]
GLOBAL SIGNAL dipw2_PinReturn $IN[526]
GLOBAL SIGNAL dipw2_IntensfPresOk $IN[527]
GLOBAL SIGNAL dipw2_HopperLowLevel $IN[528]
GLOBAL SIGNAL dipw2_FeedComplt $IN[529]
GLOBAL SIGNAL dipw2_SpearHome $IN[530]
;GLOBAL SIGNAL dipw2_Reserved $OUT[513]
;GLOBAL SIGNAL dipw2_Reserved $OUT[514]
;GLOBAL SIGNAL dipw2_Reserved $OUT[515]
;GLOBAL SIGNAL dipw2_Reserved $OUT[516]
;GLOBAL SIGNAL dipw2_Reserved $OUT[517]
GLOBAL SIGNAL dopw2_Hidraulyc_Valve $OUT[518]
GLOBAL SIGNAL dopw2_GunHome $OUT[519]
DECL GLOBAL BOOL bpw2_GunAtHome=FALSE
GLOBAL SIGNAL dopw2_GunWork $OUT[520]
DECL GLOBAL BOOL bpw2_GunAtWork=FALSE
GLOBAL SIGNAL dopw2_Nut1Intensify_Home $OUT[521]
GLOBAL SIGNAL dopw2_Nut1Intensify $OUT[522]
GLOBAL SIGNAL dopw2_StartWater $OUT[523]
GLOBAL SIGNAL dopw2_StartFeed $OUT[524]
GLOBAL SIGNAL dopw2_LevelOk $OUT[525]
GLOBAL SIGNAL dopw2_LowLevel $OUT[526]
GLOBAL SIGNAL dopw2_StepperWarningPL $OUT[527]
GLOBAL SIGNAL dopw2_EndofStepperPL $OUT[528]
GLOBAL SIGNAL dopw2_BlowOff $OUT[542]
GLOBAL SIGNAL dopw2_AdvancePin $OUT[543]
GLOBAL SIGNAL dopw2_ReturnPin $OUT[544]
GLOBAL SIGNAL dopw2_StudStripped $OUT[545]
;ENDFOLD (DNMP System 2 IO Data)
;FOLD Welder System 2 IO Data
GLOBAL SIGNAL dipw2_WeldComplete $IN[531]
GLOBAL SIGNAL dipw2_Ready $IN[532]
GLOBAL SIGNAL dipw2_Fault $IN[533]
GLOBAL SIGNAL dipw2_StepperWarning $IN[534]
GLOBAL SIGNAL dipw2_EndOfStepper $IN[535]
GLOBAL SIGNAL dipw2_StepperAreReset $IN[536]
GLOBAL SIGNAL dopw2_WeldContactEnable $OUT[529]
GLOBAL SIGNAL dopw2_WeldOnExternal $OUT[530]
GLOBAL SIGNAL dopw2_WeldInit $OUT[531]
GLOBAL SIGNAL dopw2_FaultReset $OUT[532]
GLOBAL SIGNAL dopw2_StepperReset $OUT[533]
GLOBAL SIGNAL dopw2_534SpotNumber1 $OUT[534]
GLOBAL SIGNAL dopw2_535SpotNumber2 $OUT[535]
GLOBAL SIGNAL dopw2_536SpotNumber4 $OUT[536]
GLOBAL SIGNAL dopw2_537SpotNumber8 $OUT[537]
GLOBAL SIGNAL dopw2_538SpotNumber16 $OUT[538]
GLOBAL SIGNAL dopw2_539SpotNumber32 $OUT[539]
GLOBAL SIGNAL dopw2_540SpotNumber64 $OUT[540]
GLOBAL SIGNAL dopw2_541SpotNumber128 $OUT[541]
GLOBAL SIGNAL gdopw2_SpotNumber $OUT[534]  TO $OUT[541]
;ENDFOLD (Welder System 2 IO Data)
;FOLD DNMP System 3 IO Data
;GLOBAL SIGNAL dipw3_Reserved $IN[561]
;GLOBAL SIGNAL dipw3_Reserved $IN[562]
;GLOBAL SIGNAL dipw3_Reserved $IN[563]
;GLOBAL SIGNAL dipw3_Reserved $IN[564]
;GLOBAL SIGNAL dipw3_Reserved $IN[565]
;GLOBAL SIGNAL dipw3_Reserved $IN[566]
;GLOBAL SIGNAL dipw3_Reserved $IN[567]
;GLOBAL SIGNAL dipw3_Reserved $IN[568]
GLOBAL SIGNAL dipw3_AirOK $IN[569]
GLOBAL SIGNAL dipw3_WaterOk $IN[570]
GLOBAL SIGNAL dipw3_XtfmrTempOk $IN[571]
GLOBAL SIGNAL dipw3_GunAtHome $IN[572]
GLOBAL SIGNAL dipw3_GunAtWork $IN[573]
GLOBAL SIGNAL dipw3_PinReturn $IN[574]
GLOBAL SIGNAL dipw3_IntensfPresOk $IN[575]
GLOBAL SIGNAL dipw3_HopperLowLevel $IN[576]
GLOBAL SIGNAL dipw3_FeedComplt $IN[143]
GLOBAL SIGNAL dipw3_SpearHome $IN[148]
;GLOBAL SIGNAL dipw3_Reserved $OUT[561]
;GLOBAL SIGNAL dipw3_Reserved $OUT[562]
;GLOBAL SIGNAL dipw3_Reserved $OUT[563]
;GLOBAL SIGNAL dipw3_Reserved $OUT[564]
;GLOBAL SIGNAL dipw3_Reserved $OUT[565]
GLOBAL SIGNAL dopw3_Hidraulyc_Valve $OUT[566]
GLOBAL SIGNAL dopw3_GunHome $OUT[567]
DECL GLOBAL BOOL bpw3_GunAtHome=FALSE
GLOBAL SIGNAL dopw3_GunWork $OUT[568]
DECL GLOBAL BOOL bpw3_GunAtWork=FALSE
GLOBAL SIGNAL dopw3_Nut1Intensify_Home $OUT[569]
GLOBAL SIGNAL dopw3_Nut1Intensify $OUT[570]
GLOBAL SIGNAL dopw3_StartWater $OUT[571]
GLOBAL SIGNAL dopw3_StartFeed $OUT[143]
GLOBAL SIGNAL dopw3_LevelOk $OUT[573]
GLOBAL SIGNAL dopw3_LowLevel $OUT[574]
GLOBAL SIGNAL dopw3_StepperWarningPL $OUT[575]
GLOBAL SIGNAL dopw3_EndofStepperPL $OUT[576]
GLOBAL SIGNAL dopw3_BlowOff $OUT[590]
GLOBAL SIGNAL dopw3_AdvancePin $OUT[591]
GLOBAL SIGNAL dopw3_ReturnPin $OUT[592]
GLOBAL SIGNAL dopw3_StudStripped $OUT[593]
;ENDFOLD (DNMP System 3 IO Data)
;FOLD Welder System 3 IO Data
GLOBAL SIGNAL dipw3_WeldComplete $IN[579]
GLOBAL SIGNAL dipw3_Ready $IN[580]
GLOBAL SIGNAL dipw3_Fault $IN[581]
GLOBAL SIGNAL dipw3_StepperWarning $IN[582]
GLOBAL SIGNAL dipw3_EndOfStepper $IN[583]
GLOBAL SIGNAL dipw3_StepperAreReset $IN[584]
GLOBAL SIGNAL dopw3_WeldContactEnable $OUT[577]
GLOBAL SIGNAL dopw3_WeldOnExternal $OUT[578]
GLOBAL SIGNAL dopw3_WeldInit $OUT[579]
GLOBAL SIGNAL dopw3_FaultReset $OUT[580]
GLOBAL SIGNAL dopw3_StepperReset $OUT[581]
GLOBAL SIGNAL dopw3_582SpotNumber1 $OUT[582]
GLOBAL SIGNAL dopw3_583SpotNumber2 $OUT[583]
GLOBAL SIGNAL dopw3_584SpotNumber4 $OUT[584]
GLOBAL SIGNAL dopw3_585SpotNumber8 $OUT[585]
GLOBAL SIGNAL dopw3_586SpotNumber16 $OUT[586]
GLOBAL SIGNAL dopw3_587SpotNumber32 $OUT[587]
GLOBAL SIGNAL dopw3_588SpotNumber64 $OUT[588]
GLOBAL SIGNAL dopw3_589SpotNumber128 $OUT[589]
GLOBAL SIGNAL gdopw3_SpotNumber $OUT[582]  TO $OUT[589]
;ENDFOLD (Welder System 3 IO Data)
;FOLD Nut Sensor I/O Data
GLOBAL SIGNAL aiNutSensorPW1 $IN[492]  TO $IN[505]
GLOBAL SIGNAL aiNutSensorPW2 $IN[545]  TO $IN[558]
GLOBAL SIGNAL aiNutSensorPW3 $IN[593]  TO $IN[606]
GLOBAL SIGNAL aipw1_LVDT $IN[931]  TO $IN[944]
GLOBAL SIGNAL aipw2_LVDT $IN[945]  TO $IN[958]
GLOBAL SIGNAL aipw3_LVDT $IN[959]  TO $IN[972]

GLOBAL REAL raipw1_LVDT_OPN=3400.00
GLOBAL REAL raipw2_LVDT_OPN=2600.00
GLOBAL REAL raipw3_LVDT_OPN=1260.00
GLOBAL REAL raipw1_LVDT_CLS_INV_NUT=13677.0
GLOBAL REAL raipw2_LVDT_CLS_INV_NUT=11978.0
GLOBAL REAL raipw3_LVDT_CLS_INV_NUT=10298.0
GLOBAL REAL raipw1_LVDT_CLS_W_NUT=13500.0
GLOBAL REAL raipw2_LVDT_CLS_W_NUT=13100.0
GLOBAL REAL raipw3_LVDT_CLS_W_NUT=11440.0
GLOBAL REAL raipw1_LVDT_CLS_WO_NUT=14356.0
GLOBAL REAL raipw2_LVDT_CLS_WO_NUT=13078.0
GLOBAL REAL raipw3_LVDT_CLS_WO_NUT=11483.0
GLOBAL REAL raipw1_LVDT_CLS_NO_PRT=14428.0
GLOBAL REAL raipw2_LVDT_CLS_NO_PRT=13216.0
GLOBAL REAL raipw3_LVDT_CLS_NO_PRT=11600.0
;ENDFOLD (Nut Sensor Alias I/O Data)

;FOLD 251202 New monitoring variables
GLOBAL INT iLastActiveGun=3
GLOBAL INT iSpotnr=3
GLOBAL REAL rLowerLVDT=11674.0
GLOBAL REAL rUpperLVDT=0.0
GLOBAL BOOL bGunReady2Start=FALSE
GLOBAL BOOL bDumpNutExceeded=FALSE
GLOBAL ENUM eWState Wait2Weld,FeedRequest,CloseGun,ERRORCloseGun,CheckNut,ERRORInvertedNut,ERRORNoNut,DumpNut,OpenGun,IntensifyGun,ERRORIntensifyWelder,WeldInitiate,GunHome
DECL GLOBAL eWState eCurrentState=#GunHome
;ENDFOLD

ENDDAT
